Fanuc TP program (LS listing): unbalanced_bracket.ls

/PROG  UNBAL
/ATTR
OWNER		= MNEDITOR;
COMMENT		= "";
PROG_SIZE	= 100;
CREATE		= DATE 25-01-01  TIME 00:00:00;
MODIFIED	= DATE 25-01-01  TIME 00:00:00;
FILE_NAME	= ;
VERSION		= 0;
LINE_COUNT	= 2;
MEMORY_SIZE	= 100;
PROTECT		= READ_WRITE;
TCD:  STACK_SIZE	= 0,
      TASK_PRIORITY	= 50,
      TIME_SLICE	= 0,
      BUSY_LAMP_OFF	= 0,
      ABORT_REQUEST	= 0,
      PAUSE_REQUEST	= 0;
DEFAULT_GROUP	= 1,*,*,*,*;
CONTROL_CODE	= 00000000 00000000;
/APPL
/MN
   1:  R[1]=R[2+R[3] ;
   2:   ;
/POS
/END
